SYMBOL_TABLE
"Constants_RSM"	DB 1	DB 1	// Sheet 2 (RSM)
"HISIGMTR-VALs"	DB 2	DB 2
"LOSIGMTR-VALs"	DB 3	DB 3
"AIN_VALs_VIB"	DB 4	FB 1	// DB for analog vibration inputs
"GAINBI-VALs"	DB 5	DB 5
"DELTAW-VALs"	DB 6	DB 6	// DELTAW contants
"HILOLMTV-VALs"	DB 7	DB 7
"HILOMTR-VALs"	DB 8	DB 8
"AVALGEN"	DB 9	DB 9	// Analog Value Generation
"DVALGEN"	DB 10	DB 10	// Digital Value Generation
"RUNAVG_VALs_369_370"	DB 11	FB 2	// RUNAVG_DB for blocks 369  and 370
"HISIGMTV-VALs"	DB 12	DB 12
"LOSIGMTV-VALs"	DB 13	DB 13
"XLIMIT_VALs"	DB 14	DB 14
"AIFCTGEN_Vals"	DB 15	DB 15
"MULTGB_VALs"	DB 16	DB 16
"SUM2W_VALs"	DB 17	DB 17
"RATEMTR_VALs"	DB 18	DB 18
"XSUM_VALs"	DB 19	DB 19
"XTRANSF_VALs"	DB 20	DB 20
"XHISEL_VALs"	DB 21	DB 21
"AIN_VALs_TEMP_100"	DB 22	FB 1
"DIVIDEGB_VALs"	DB 23	DB 23
"AIN_VALs_TEMP_286"	DB 24	FB 1
"POLY_VALs"	DB 25	DB 25
"SUM4W_VALs"	DB 26	DB 26
"SUM8W_VALs"	DB 27	DB 27
"AIN_VALs_TEMP_661"	DB 28	FB 1	// DB for analog temperature inputs
"AIN_VALs_PRESS_760"	DB 29	FB 1	// DB for pressure analog inputs
"RESETSUM_VALs"	DB 30	DB 30
"AIN_VALs_POS_25"	DB 31	FB 1
"XMULT_VALs"	DB 32	DB 32
"ATCTime_VALs"	DB 33	DB 33	// Time declaration for all the timers used
"DIGCNTNF_VALs"	DB 34	DB 34
"Constants_ATC"	DB 35	DB 35
"RUNAVG_VALs_235"	DB 36	FB 2
"AIN_VALs_POS_2"	DB 37	FB 1	// DB for analog position inputs
"RSMTime_VALs"	DB 38	DB 38
"TIMECHG_VALs"	DB 39	DB 39
"AIN"	FB 1	FB 1	// REAL conversion of analog input signals
"RUNAVG"	FB 2	FB 2	// Average of time based samples of input
"DRUMD16"	FB 3	FB 3	// Drum Controller with Sixteen Digital Outputs
"QC"	FC 1	FC 1	// QCHK1BAD
"Sheet 24 (ATC)"	FC 2	FC 2	// VIBRATION MONITOR
"TOD_Conversion"	FC 3	FC 3	// Supporting Block for Sheet 24 (ATC)
"Sheet 2 (RSM)"	FC 4	FC 4	// Initialization of constants in sheet 2 (RSM)
"TRANSF"	FC 5	FC 5	// Transfer between Two Analog Inputs
"AIFCTGEN"	FC 6	FC 6
"BIN_SEARCH"	FC 7	FC 7
"XHISEL"	FC 8	FC 8	// Selects the Greater of Two Gained and Biased Inputs
"QAVGN"	FC 10	FC 10	// Average up to Eight Analog Points
"HISIGMTR"	FC 11	FC 11	// High Signal Monitor with Reset Deadband and Fixed Limit
"LOSIGMTR"	FC 12	FC 12	// Low Signal Monitor with Reset Deadband and Fixed Limit
"GAINBI"	FC 14	FC 14	// Gain and Bias an Input
"DELTAW"	FC 15	FC 15	// Difference between Two Weighted Inputs
"HILOLMTV"	FC 16	FC 16	// High/Low Limiter, Variable Limits
"HILOMTR"	FC 18	FC 18	// High/Low Signal Monitor with Reset Deadband and Fixed Limits
"QTRANSN"	FC 19	FC 19	// Automatic transfer between analog inputs, select best quality
"DIVIDEGB"	FC 21	FC 21	// Divider with Gain and Bias
"POLY"	FC 22	FC 22	// Fifth Order Polynomial Equation
"QBLOCK"	FC 23	FC 23	// Output is equal to input and output quality is good.
"SUM8W"	FC 24	FC 24
"Sheet 3 (RSM)"	FC 25	FC 25	// FSST & TIMP & TSAT (Analog)
"Sheet 4 (RSM)"	FC 26	FC 26	// HP FILM & TICM & TMAX (Analog)
"Sheet 5 (RSM)"	FC 27	FC 27	// MWINC LOGIC (Digital)
"Sheet 7 (RSM)"	FC 28	FC 28	// HP INVALID LOGIC (Digital)
"RESETSUM"	FC 29	FC 29	// Summer with Reset
"Sheet 6 (RSM)"	FC 30	FC 30	// HP Stress Counters (Analog)
"HISIGMTV"	FC 31	FC 31	// High Signal Monitor, Reset Deadband and Variable Limits
"LOSIGMTV"	FC 32	FC 32	// Low Signal Monitor, Reset Deadband, Variable Limit
"HISEL10"	FC 33	FC 33	// High Signal Selector with 'TWO' Inputs
"XLIMIT"	FC 34	FC 34	// Limits a Gained and Biased Input
"LOSEL10"	FC 35	FC 35	// Low Signal Selector with 'TWO' Inputs
"Sheet 9 (RSM)"	FC 36	FC 36	// HP ROTSURF, T1-5 & TP1-4 (Analog)
"Sheet 8 (RSM)"	FC 37	FC 37	// HXFER & TWC (Analog)
"Sheet 10 (RSM)"	FC 38	FC 38	// HP TEMP T6-T15 (Analog)
"Sheet11 (RSM)"	FC 39	FC 39	// HP TEMP T16-T23 (Analog)
"MULTGB"	FC 40	FC 40	// Multiplier with Gain and Bias
"SUM2W"	FC 41	FC 41	// Sum of Two Weighted Inputs
"RATEMTR"	FC 42	FC 42	// Rate of Change Monitor, Reset Deadband, Fixed Rate Limit
"XSUM"	FC 43	FC 43	// Add Two Gained and Biased Inputs
"XTRANSF"	FC 44	FC 44	// Select a Gained and Biased Input Based on a Flag
"Sheet 12 (RSM)"	FC 45	FC 45	// HP TAVG (Analog)
"Sheet 13 (RSM)"	FC 46	FC 46	// HP EFFECTIVE TEMP DIFF. (Analog)
"Sheet 14 (RSM)"	FC 47	FC 47	// HP DRUM TIMERS (Analog)
"Sheet 15 (RSM)"	FC 48	FC 48	// HP TD1FT1-15 (Analog)
"Sheet 16 (RSM)"	FC 51	FC 51	// HP ANTIC. DIFF. (Analog)
"Sheet 17 (RSM)"	FC 53	FC 53	// % ROTOR STRESS LIMIT (Analog)
"XMULT"	FC 54	FC 54	// Multiples Two Gained and Biased Inputs
"Sheet 18 (RSM)"	FC 55	FC 55	// SMW INC/DEC (Analog)
"Sheet 19 (RSM)"	FC 57	FC 57	// TBP (Analog)
"Sheet 20 (RSM)"	FC 58	FC 58	// MWINCR (Analog)
"Sheet 21 (RSM)"	FC 59	FC 59	// ATC RATE & LOAD RESERVE (Analog)
"SUM4W"	FC 60	FC 60
"Sheet 22 (RSM)"	FC 61	FC 61	// REQ. STM CHEST METAL TEMP (Analog)
"Sheet 23 (RSM)"	FC 62	FC 62	// HP ROTOR STRESS LIMIT (Digital)
"Sheet 24 (RSM)"	FC 63	FC 63	// ATC TARGET (Analog)
"Sheet 25 (RSM)"	FC 64	FC 64	// TRANSFER DELAY (Digital)
"Sheet 26 (RSM)"	FC 65	FC 65	// LADDERS 35, 128, RESONANCE RANGE LOGIC (Digital)
"Sheet 28 (RSM)"	FC 66	FC 66	// LADDERS 22, 500, 600, DIGITAL POINTERS TMAX & TWC LOGIC (Digital)
"Sheet 29 (RSM)"	FC 67	FC 67	// LADDERS 29, 31, 500, FIRST STAGE STM > 75 *C (Digital)
"Sheet 27 (RSM)"	FC 68	FC 68	// LADDERS 43, 129, RTSHOLD (Digital)
"Sheet 30 (RSM)"	FC 69	FC 69	// LADDER 126, SYNC LOGIC & OVERRIDE (Digital)
"Sheet 31 (RSM)"	FC 70	FC 70	// LADDER 33, ANTIC HP STRESS > LIMIT (Digital)
"Sheet 32 (RSM)"	FC 71	FC 71	// LADDERS 37, 125, 130, SYNC LOGIC & OVERRIDE (Digital)
"Sheet 33 (RSM)"	FC 72	FC 72	// LADDER 124, 127, SYNC LOGIC & TVGVINIT (Digital)
"Sheet 34 (RSM)"	FC 73	FC 73	// LADDERS 122, 123, 135, SET SPEED PLATEAU (Digital)
"Sheet 35 (RSM)"	FC 74	FC 74	// LADDER 120, 121, P15 ALARMS ESTIMATE ROLL TIME LOGIC & ATC VPL (Digital)
"Sheet 36 (RSM)"	FC 75	FC 75	// LADDER 41, 119, P15 ALARMS (Digital)
"Sheet 37 (RSM)"	FC 76	FC 76	// GENERATOR AND EXCITOR TEMPERATURES (Analog)
"Sheet 2 (ATC)"	FC 77	FC 77	// LADDER 500, SENSOR FAIL (Digital)
"Sheet 3 (ATC)"	FC 78	FC 78	// SENSOR FAIL (Digital)
"DIGCNTNF"	FC 79	FC 79	// Digital Counter with Flag
"Sheet 4 (ATC)"	FC 81	FC 81	// LADDERS 1, 3 (Digital)
"Sheet 5 (ATC)"	FC 82	FC 82	// LADDERS 3, 5, 9, 600, P00M01-M11 (Digital)
"Sheet 6 (ATC)"	FC 83	FC 83	// LADDERS 7, 9, 13, ATC PERMISSIVE (Digital)
"Sheet 7 (ATC)"	FC 84	FC 84	// LADDER 81. LOOPS 27, 33. WATER COOLED GENERATOR (Analog)
"Sheet 8 (ATC)"	FC 85	FC 85	// LADDERS 91, 108, 133, GENERATOR ANNUNCIATOR (Digital)
"Sheet 9 (ATC)"	FC 86	FC 86	// LADDERS 81,83,85,87,109,130. LOOPS 28-30. EXMON & COOLGSHI & P09MXX  (Digital)
"Sheet 10 (ATC)"	FC 87	FC 87	// LADDERS 31, 34, 36, GENERATOR CALCULATIONS (Analog)
"Sheet 11 (ATC)"	FC 88	FC 88	// LADDERS 15, 17, 18. LOOPS 2, 3. STEAM CHEST - OIL COOLER MONITOR (Analog)
"2xHISIGMTV, QC"	FC 89	FC 89	// Supporting block for sheet 12, 24 (ATC)
"Sheet 12 (ATC)"	FC 91	FC 91	// BEARING METAL TEMPERATURES (Analog)
"Sheet 13 (ATC)"	FC 92	FC 92	// BEARING METAL, OIL COOLER - P08MXX (Digital)
"Sheet 14 (ATC)"	FC 93	FC 93	// BEARING METAL - P08M05, 8 (Digital)
"Sheet 15 (ATC)"	FC 94	FC 94	// ROTOR POSITION, DIFF EXPANSION (Analog)
"Sheet 16 (ATC)"	FC 95	FC 95	// ROTOR POSITION DIFFERENTIAL EXPANSION P11MXX (Digital)
"Sheet 17 (ATC)"	FC 96	FC 96	// LOOPS 39, 40, 41. CONDENSOR PRESS LP EXH HOOD (Analog)
"Sheet 18 (ATC)"	FC 97	FC 97	// LADDERS 89, 90, 189, 190. GLAND, EXH, VAC - P10MXX (Digital)
"Sheet 19 (ATC)"	FC 98	FC 98	// BRG TEMPERATURE HIGH & VBINC (Digital)
"Sheet 20 (ATC)"	FC 99	FC 99	// VIBRATION LIMIT (Analog)
"Sheet 21 (ATC)"	FC 100	FC 100	// LADDERS 302,304,306,400. VIBRATION ALARM AND TRIP (Digital)
"Sheet 22 (ATC)"	FC 101	FC 101	// LADDERS 32, 33, 41. VIBRATION RUNUP / RUNDOWN LOGIC (Digital)
"Sheet 23 (ATC)"	FC 102	FC 102	// LADDER 39. VIBRATION RUNDOWN / RUNBACK LOGIC (Digital)
"3xHISIGMTV, 1xLOSIGMTV"	FC 103	FC 103
"3xLOSIGMTV, 1xHISIGMTV"	FC 104	FC 104
"SCALE"	FC 105	FC 105	// Scaling Values
"Sheet 25 (ATC)"	FC 106	FC 106	// SPEED RESONANT RANGE MONITOR (Analog)
"Sheet 26 (ATC)"	FC 107	FC 107	// LADDERS 150, 420. VIBRATION SPEED REF LOGIC (Digital)
"Sheet 27 (ATC)"	FC 108	FC 108	// VIBRATION RUNBACK SPEED REF (Analog)
"Sheet 28 (ATC)"	FC 109	FC 109	// LADDERS 30, 43, 307, 308, 309. VIBRATION RUNUP/RUNTHRU LOGIC (Digital)
"Sheet 29 (ATC)"	FC 110	FC 110	// VIBRATION RUN THRU REF (Analog)
"Sheet 30 (ATC)"	FC 111	FC 111	// VIBRATION SPEED REF (Analog)
"Sheet 31 (ATC)"	FC 112	FC 112	// LOOPS 18, 19. WATER DETECTION (Analog)
"Sheet 32 (ATC)"	FC 113	FC 113	// LADDERS 49, 51, 53. DRAIN VALVE LOGIC (Digital)
"DT_TOD"	FC 115	FC 115	// DT to TOD
"SUBB24"	FC 116	FC 116	// Supporting block for sheet 24 (ATC)
"TIMECHG"	FC 117	FC 117	// Check Real-Time Clock, Set Flags
"Sheet 33 (ATC)"	FC 118	FC 118	// LOOPS 4, 5 (Analog)
"Sheet 34 (ATC)"	FC 119	FC 119	// LADDERS 19, 21, 23, 25, 27. TURNING GEAR - P03MXX (Digital)
"Sheet 35 (ATC)"	FC 120	FC 120	// LOOPS 6, 60. THRUST BEARING, ROTOR ECCEN. (Analog)
"Sheet 36 (ATC)"	FC 121	FC 121	// LADDERS 27, 600. ATC PLATEAU FLAGS (Digital)
"Sheet 37 (ATC)"	FC 122	FC 122	// OVERRIDE LOGIC (Analog)
"Sheet 38 (ATC)"	FC 123	FC 123	// OVERRIDE LOGIC (Digital)
"Sheet 39 (ATC)"	FC 124	FC 124	// OVERRIDE LOGIC (Digital)
"Sheet 40 (ATC)"	FC 125	FC 125	// LADDERS 200, 201, 203, 220. REQUEST TRIP P07MXX (Digital)
"Sheet 41 (ATC)"	FC 126	FC 126	// LADDERS 201, 202, 203. HOLD 1 & 2 - P07M13 (Digital)
"Sheet 42 (ATC)"	FC 127	FC 127	// LADDERS 110, 111, 112, 113. OVERRIDE & P07M12 (Digital)
"Sheet 43 (ATC)"	FC 128	FC 128	// LADDERS 11, 113, 114. HOLD LOAD & P07M09 - 14 (Digital)
"Sheet 44 (ATC)"	FC 129	FC 129	// LADDERS 115, 116. HOLD WS & P07M02 - 04 (Digital)
"Sheet 45 (ATC)"	FC 130	FC 130	// LADDERS 117, 118. LOAD RATE INC/DEC P07M05 - 08 (Digital)
"Sheet 47 (ATC)"	FC 131	FC 131	// LADDERS 118, 192. P00M00A-G (Digital)
"Sheet 46 (ATC)"	FC 132	FC 132	// LOOPS 63, 65. LOAD RATE (Analog)
"Sheet 48_49 (ATC)"	FC 133	FC 133	// Initialization of ATC constants from AVALGEN DB
"ASSAP"	I 0.0	BOOL	//  (ATC) - (FieldIO4-M1)
"BOPL"	I 0.1	BOOL	//  (ATC) - (FieldIO4-M1)
"BVAP"	I 0.2	BOOL	//  (ATC) - (FieldIO4-M1)
"DVSAP"	I 0.3	BOOL	//  (ATC) - (FieldIO4-M1)
"EHFPL"	I 0.4	BOOL	//  (ATC) - (FieldIO4-M1)
"EHSO"	I 0.5	BOOL	//  (ATC) - (FieldIO4-M1)
"GDOGF"	I 0.6	BOOL	//  (ATC) - (FieldIO4-M1)
"GVRNLV"	I 0.7	BOOL	//  (ATC) - (FieldIO4-M1)
"HPDVC"	I 1.0	BOOL	//  (ATC) - (FieldIO4-M1)
"HPDVO"	I 1.1	BOOL	//  (ATC) - (FieldIO4-M1)
"MBCSU"	I 1.2	BOOL	//  (ATC) - (FieldIO4-M1)
"MELIT"	I 1.3	BOOL	//  (ATC) - (FieldIO4-M1)
"MVHPIT"	I 1.4	BOOL	//  (ATC) - (FieldIO4-M1)
"OEPIT"	I 1.5	BOOL	//  (ATC) - (FieldIO4-M1)
"RSBC"	I 1.6	BOOL	//  (ATC) - (FieldIO4-M1)
"RSBSU"	I 1.7	BOOL	//  (ATC) - (FieldIO4-M1)
"TGE"	I 2.0	BOOL	//  (ATC) - (FieldIO5-M1)
"VRO"	I 2.1	BOOL	//  (ATC) - (FieldIO5-M1)
"VROUS"	I 2.2	BOOL	//  (ATC) - (FieldIO5-M1)
"VRSOTP"	I 2.3	BOOL	//  (ATC) - (FieldIO5-M1)
"CAB4T1"	IW 512	WORD	//  (RSM) - (FieldIO4-M3)
"CNDP1"	IW 514	WORD	//  (RSM) - (FieldIO4-M3)
"FSST1"	IW 516	WORD	//  (RSM) - (FieldIO4-M3)
"B1T1"	IW 518	WORD	//  (ATC) - (FieldIO4-M3)
"B2T1"	IW 520	WORD	//  (ATC) - (FieldIO4-M3)
"B3T1"	IW 522	WORD	//  (ATC) - (FieldIO4-M3)
"B4T1"	IW 524	WORD	//  (ATC) - (FieldIO4-M3)
"B5T1"	IW 526	WORD	//  (ATC) - (FieldIO4-M3)
"B6T1"	IW 528	WORD	//  (ATC) - (FieldIO4-M4)
"RP1"	IW 530	WORD	//  (ATC) - (FieldIO4-M4)
"TBFCT1"	IW 532	WORD	//  (ATC) - (FieldIO4-M4)
"TBFLT1"	IW 534	WORD	//  (ATC) - (FieldIO4-M4)
"TBRCT1"	IW 536	WORD	//  (ATC) - (FieldIO4-M4)
"TBRLT1"	IW 538	WORD	//  (ATC) - (FieldIO4-M4)
"VB9"	IW 540	WORD	//  (ATC) - (FieldIO4-M4)
"FSMT1"	IW 542	WORD	//  (RSM) - (FieldIO4-M4)
"B7T"	IW 544	WORD	//  (ATC) - (FieldIO4-M5)
"B8T"	IW 546	WORD	//  (ATC) - (FieldIO4-M5)
"B9T"	IW 548	WORD	//  (ATC) - (FieldIO4-M5)
"B10T"	IW 550	WORD	//  (ATC) - (FieldIO4-M5)
"CAB5T1"	IW 552	WORD	//  (ATC) - (FieldIO4-M5)
"CAB5T2"	IW 554	WORD	//  (ATC) - (FieldIO4-M5)
"CASEXP"	IW 556	WORD	//  (ATC) - (FieldIO4-M5)
"DEGEN"	IW 558	WORD	//  (ATC) - (FieldIO4-M5)
"VB1"	IW 560	WORD	//  (ATC) - (FieldIO4-M6)
"VB2"	IW 562	WORD	//  (ATC) - (FieldIO4-M6)
"VB3"	IW 564	WORD	//  (ATC) - (FieldIO4-M6)
"VB4"	IW 566	WORD	//  (ATC) - (FieldIO4-M6)
"VB5"	IW 568	WORD	//  (ATC) - (FieldIO4-M6)
"VB6"	IW 570	WORD	//  (ATC) - (FieldIO4-M6)
"VB7"	IW 572	WORD	//  (ATC) - (FieldIO4-M6)
"VB8"	IW 574	WORD	//  (ATC) - (FieldIO4-M6)
"CAB4T2"	IW 576	WORD	//  (RSM) - (FieldIO5-M3)
"CNDP2"	IW 578	WORD	//  (RSM) - (FieldIO5-M3)
"FSST2"	IW 580	WORD	//  (RSM) - (FieldIO5-M3)
"B1T2"	IW 582	WORD	//  (ATC) - (FieldIO5-M3)
"B2T2"	IW 584	WORD	//  (ATC) - (FieldIO5-M3)
"B3T2"	IW 586	WORD	//  (ATC) - (FieldIO5-M3)
"B4T2"	IW 588	WORD	//  (ATC) - (FieldIO5-M3)
"B5T2"	IW 590	WORD	//  (ATC) - (FieldIO5-M3)
"B6T2"	IW 592	WORD	//  (ATC) - (FieldIO5-M4)
"RP2"	IW 594	WORD	//  (ATC) - (FieldIO5-M4)
"TBFCT2"	IW 596	WORD	//  (ATC) - (FieldIO5-M4)
"TBFLT2"	IW 598	WORD	//  (ATC) - (FieldIO5-M4)
"TBRCT2"	IW 600	WORD	//  (ATC) - (FieldIO5-M4)
"TBRLT2"	IW 602	WORD	//  (ATC) - (FieldIO5-M4)
"VB10"	IW 604	WORD	//  (ATC) - (FieldIO5-M4)
"LPGST"	IW 606	WORD	//  (RSM) - (FieldIO5-M4)
"EHFLT"	IW 608	WORD	//  (ATC) - (FieldIO5-M5)
"HPBMIDT"	IW 610	WORD	//  (ATC) - (FieldIO5-M5)
"HPCMIDT"	IW 612	WORD	//  (ATC) - (FieldIO5-M5)
"LP1GNT"	IW 614	WORD	//  (ATC) - (FieldIO5-M5)
"LP1GVT"	IW 616	WORD	//  (ATC) - (FieldIO5-M5)
"LP2GNT"	IW 618	WORD	//  (ATC) - (FieldIO5-M5)
"LP2GVT"	IW 620	WORD	//  (ATC) - (FieldIO5-M5)
"ROTECC"	IW 622	WORD	//  (ATC) - (FieldIO5-M5)
"OCIT"	IW 624	WORD	//  (RSM) - (FieldIO5-M6)
"OCOT"	IW 626	WORD	//  (RSM) - (FieldIO5-M6)
"Main program routine"	OB 1	OB 1
"I/O_FLT1"	OB 82	OB 82	// I/O Point Fault 1
"I/O_FLT2"	OB 83	OB 83	// I/O Point Fault 2
"OBNL_FLT"	OB 85	OB 85	// OB Not Loaded Fault
"RACK_FLT"	OB 86	OB 86	// Loss of Rack Fault
"COMPLETE RESTART"	OB 100	OB 100	// Complete Restart
"PROG_ERR"	OB 121	OB 121	// Programming Error
"MOD_ERR"	OB 122	OB 122	// Module Access Error
"ATCALO"	Q 0.0	BOOL	//  (ATC) - (FieldIO4-M2)
"ATCASSO"	Q 0.1	BOOL	//  (ATC) - (FieldIO4-M2)
"ATCMEO"	Q 0.2	BOOL	//  (ATC) - (FieldIO4-M2)
"ATCNAO"	Q 0.3	BOOL	//  (ATC) - (FieldIO4-M2)
"ATCSMO"	Q 0.4	BOOL	//  (ATC) - (FieldIO4-M2)
"ATCTAO"	Q 0.5	BOOL	//  (ATC) - (FieldIO4-M2)
"ATCTO"	Q 0.6	BOOL	//  (ATC) - (FieldIO4-M2)
"CHPDVO"	Q 0.7	BOOL	//  (ATC) - (FieldIO4-M2)
"CRSBO"	Q 1.0	BOOL	//  (ATC) - (FieldIO4-M2)
"LPHTO"	Q 1.1	BOOL	//  (ATC) - (FieldIO4-M2)
"LPVHTO"	Q 1.2	BOOL	//  (ATC) - (FieldIO4-M2)
"WDHTO"	Q 1.3	BOOL	//  (ATC) - (FieldIO4-M2)
"WDVHTO"	Q 1.4	BOOL	//  (ATC) - (FieldIO4-M2)
"RSINV1"	Q 2.0	BOOL	//  (RSM) - (FieldIO5-M2)
"RSINV2"	Q 2.1	BOOL	//  (RSM) - (FieldIO5-M2)
"RSMON1"	Q 2.2	BOOL	//  (RSM) - (FieldIO5-M2)
"RSMON2"	Q 2.3	BOOL	//  (RSM) - (FieldIO5-M2)
"RSSENO"	Q 2.4	BOOL	//  (RSM) - (FieldIO5-M2)
"SPHLD"	Q 2.5	BOOL	//  (RSM) - (FieldIO5-M2)
"READ_CLK"	SFC 1	SFC 1	// Read System Clock
"TIME_TCK"	SFC 64	SFC 64	// Read the System Time
"HISIGMTR-UDT"	UDT 1	UDT 1
"LOSIGMTR-UDT"	UDT 2	UDT 2
"DBEQUALS-UDT"	UDT 3	UDT 3
"GAINBI-UDT"	UDT 4	UDT 4
"DELTAW-UDT"	UDT 5	UDT 5
"HILOLMTV-UDT"	UDT 6	UDT 6	// constants for HILOLMTV
"HILOMTR-UDT"	UDT 7	UDT 7
"HISIGMTV-UDT"	UDT 8	UDT 8
"LOSIGMTV-UDT"	UDT 9	UDT 9
"XLIMIT-UDT"	UDT 10	UDT 10
"MULTGB-UDT"	UDT 11	UDT 11
"SUM2W-UDT"	UDT 12	UDT 12
"RATEMTR-UDT"	UDT 13	UDT 13
"XSUM-UDT"	UDT 14	UDT 14
"XTRANSF-UDT"	UDT 15	UDT 15
"XHISEL_UDT"	UDT 16	UDT 16
"TRKHOLD-UDT"	UDT 18	UDT 18
"SUM4W-UDT"	UDT 20	UDT 20
"AIFCTGEN_UDT"	UDT 21	UDT 21
"DIVIDEGB_UDT"	UDT 22	UDT 22
"POLY_UDT"	UDT 23	UDT 23
"SUM8W_UDT"	UDT 24	UDT 24
"RESETSUM_UDT"	UDT 25	UDT 25
"XMULT_UDT"	UDT 26	UDT 26
"DIGCNTNF_UDT"	UDT 27	UDT 27
"TIMECHG_UDT"	UDT 28	UDT 28
"VAT (ATC-RSM)"	VAT 1	
END_SYMBOL_TABLE
